FUNCTION IsValidLink : BOOL
VAR_INPUT
	Link : I_Link;
END_VAR

IsValidLink := Link <> 0;

END_FUNCTION

(* stored: Version 1.1.0.1, ProductVersion 3.1.4024.12
   POU IsValidLink: Id {eac2773c-30ae-0cc3-3642-973a7d951e52}, SpecialFunc None *)
